FUNCTION_BLOCK I_MSS (* Machine Selected Speed MSS *)
  (* Standard: ISO 11783-7; Classification: PGN 65097; Function: Machine Selected Speed MSS; Description: Copyright (c) 2024 HR Agrartechnik GmbH This program and the accompanying materials are made available under the terms of the Eclipse Public License 2.0 which is available at https://www.eclipse.org/legal/epl-2.0/ SPDX-License-Identifier: EPL-2.0 Message that provides the current machine selected speed, direction and source parameters. https://www.isobus.net/isobus/pGNAndSPN/2233?type=PGN *)
  (* Version 1.0, 2024-07-09, Franz Hoepfinger, HR Agrartechnik GmbH *)
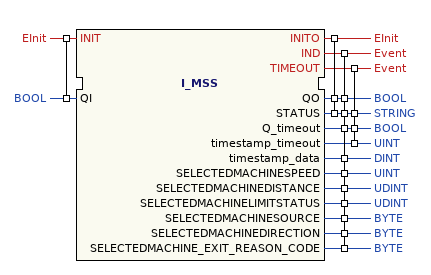
  EVENT_INPUT
    INIT : EInit WITH QI; (* Service Initialization *)
  END_EVENT
  EVENT_OUTPUT
    INITO : EInit WITH QO, STATUS; (* Initialization Confirm *)
    IND WITH QO, timestamp_data, STATUS, Q_timeout, SELECTEDMACHINESPEED, SELECTEDMACHINEDISTANCE, SELECTEDMACHINELIMITSTATUS, SELECTEDMACHINESOURCE, SELECTEDMACHINEDIRECTION, SELECTEDMACHINE_EXIT_REASON_CODE; (* Indication from Resource *)
    TIMEOUT WITH timestamp_timeout, STATUS, Q_timeout;
  END_EVENT
  VAR_INPUT
    QI : BOOL; (* Event Input Qualifier *)
  END_VAR
  VAR_OUTPUT
    QO : BOOL; (* Event Output Qualifier *)
    STATUS : STRING;
    Q_timeout : BOOL;
    timestamp_timeout : UINT;
    timestamp_data : DINT;
    SELECTEDMACHINESPEED : UINT; (* Machine selected speed (see Attributes for Details) *) {SET_ATTRIBUTE(SPN, 4305)} {SET_ATTRIBUTE(SP_Name, 'Machine selected speed')} {SET_ATTRIBUTE(SP_Position_In_PG, '1-2')} {SET_ATTRIBUTE(SP_Length, 16)} (* 16 bits *) {SET_ATTRIBUTE(Scaling, '0.001 m/s/bit, upper byte 0.256 m/s/bit')} {SET_ATTRIBUTE(Offset, )} {SET_ATTRIBUTE(Link, 'https://www.isobus.net/isobus/pGNAndSPN/2232?type=SPN')}
    SELECTEDMACHINEDISTANCE : UDINT; (* Machine selected distance (see Attributes for Details) *) {SET_ATTRIBUTE(SPN, 4306)} {SET_ATTRIBUTE(SP_Name, 'Machine selected distance')} {SET_ATTRIBUTE(SP_Position_In_PG, '3-6')} {SET_ATTRIBUTE(SP_Length, 32)} (* 32 bits *) {SET_ATTRIBUTE(Scaling, '0.001 m/bit')} {SET_ATTRIBUTE(Offset, )} {SET_ATTRIBUTE(Link, 'https://www.isobus.net/isobus/pGNAndSPN/2233?type=SPN')}
    SELECTEDMACHINELIMITSTATUS : UDINT; (* Machine selected speed limit status *) {SET_ATTRIBUTE(SPN, 4307)} {SET_ATTRIBUTE(SP_Name, 'Machine selected speed limit status')} {SET_ATTRIBUTE(SP_Position_In_PG, '8.6')} {SET_ATTRIBUTE(SP_Length, 3)} (* 3 bits *) {SET_ATTRIBUTE(Scaling, '8 states/3 bit')} {SET_ATTRIBUTE(Offset, )} {SET_ATTRIBUTE(Link, 'https://www.isobus.net/isobus/pGNAndSPN/2230?type=SPN')}
    SELECTEDMACHINESOURCE : BYTE; (* Machine selected speed source *) {SET_ATTRIBUTE(SPN, 4308)} {SET_ATTRIBUTE(SP_Name, 'Machine selected speed source')} {SET_ATTRIBUTE(SP_Position_In_PG, '8.3')} {SET_ATTRIBUTE(SP_Length, 3)} (* 3 bits *) {SET_ATTRIBUTE(Scaling, '8 states/3 bit')} {SET_ATTRIBUTE(Offset, )} {SET_ATTRIBUTE(Link, 'https://www.isobus.net/isobus/pGNAndSPN/2229?type=SPN')}
    SELECTEDMACHINEDIRECTION : BYTE; (* Machine selected direction (see Attributes for Details) *) {SET_ATTRIBUTE(SPN, 4309)} {SET_ATTRIBUTE(SP_Name, 'Machine selected direction')} {SET_ATTRIBUTE(SP_Position_In_PG, '8.1')} {SET_ATTRIBUTE(SP_Length, 2)} (* 2 bits *) {SET_ATTRIBUTE(Scaling, '4 states/2 bit')} {SET_ATTRIBUTE(Offset, )} {SET_ATTRIBUTE(Link, 'https://www.isobus.net/isobus/pGNAndSPN/2228?type=SPN')}
    SELECTEDMACHINE_EXIT_REASON_CODE : BYTE; (* Machine selected speed exit/reason code *) {SET_ATTRIBUTE(SPN, 5818)} {SET_ATTRIBUTE(SP_Name, 'Machine selected speed exit/reason code')} {SET_ATTRIBUTE(SP_Position_In_PG, '7.1')} {SET_ATTRIBUTE(SP_Length, 6)} (* 6 bits *) {SET_ATTRIBUTE(Scaling, '64 states/6 bit')} {SET_ATTRIBUTE(Offset, )} {SET_ATTRIBUTE(Link, 'https://www.isobus.net/isobus/pGNAndSPN/2231?type=SPN')}
  END_VAR
END_FUNCTION_BLOCK
